FUNCTION_BLOCK PUB_2
  (* Standard: 61499-2 *)
  (* Version 10-09-13, slimrte *)
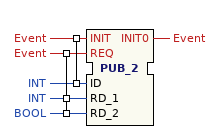
  EVENT_INPUT
    INIT WITH ID;
    REQ WITH RD_1, RD_2;
  END_EVENT
  EVENT_OUTPUT
    INIT0;
  END_EVENT
  VAR_INPUT
    ID : INT;
    RD_1 : INT;
    RD_2 : BOOL;
  END_VAR
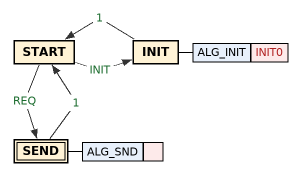
  EC_STATES
    SEND : ALG_SND;
    START;
    INIT : ALG_INIT -> INIT0;
  END_STATES
  EC_TRANSITIONS
    START TO INIT := INIT;
    START TO SEND := REQ;
    SEND TO START := 1;
    INIT TO START := 1;
  END_TRANSITIONS
  ALGORITHM ALG_SND IN Lua:
IF (NOT(RD_1_ = RD_1)) OR (NOT(RD_2_ = RD_2)) THEN
      ASM
	    LOAD RD_1
	    LOAD RD_2
	    CONST 2
	    LOAD ID
	    NISND
	  END_ASM
	  RD_1_ := RD_1;
	  RD_2_ := RD_2;
	END_IF;
  END_ALGORITHM
  ALGORITHM ALG_INIT IN Lua:

  END_ALGORITHM
END_FUNCTION_BLOCK
